FUNCTION_BLOCK FB_WinderSpeedControl
VAR_INPUT
    //==============================================================
    // ─────────────── MODE SELECTION / REFERENCES ───────────────
    //==============================================================
    groupSpeedAutoMan          : BOOL;  // TRUE = Auto, FALSE = Manual
    enableTorqueControl          : BOOL;  // TRUE = Auto, FALSE = Manual

    groupAutoSpeedMPM          : REAL;  // Auto speed reference [m/min]
    groupManualSpeedMPM        : REAL;  // Manual speed reference [m/min]
    groupRecoverSpeedCmd       : BOOL;  // Recover (temporary speed bump)
    groupRecoverIncrement      : REAL;  // Recover increment [m/min]

	
	torqueFeedback				: REAL;
    //==============================================================
    // ─────────────── DIAMETERS (mm) ───────────────
    //==============================================================
    diameter       : REAL;  // Diameter of group 1 master

    //==============================================================
    // ─────────────── CONFIGURATION / LIMITS ───────────────
    //==============================================================
    groupMasterMaxSpeedRPM     : REAL;  		// Max allowed master RPM
    rampUpRate					: REAL := 0.1;  // Ramp acceleration [RPM/s]
    rampDownRate				: REAL := 0.1;  // Ramp acceleration [RPM/s]
	
    state                      : INT;   // Machine state (5 = STOPPING)

    groupSpeedDifInc           : BOOL;  // Increment group speed offset
    groupSpeedDifDec           : BOOL;  // Decrement group speed offset
    groupSpeedDifLimLow        : REAL;  // Min offset [%]
    groupSpeedDifLimHigh       : REAL;  // Max offset [%]

    rampReset                  : BOOL;  // Reset ramp command
	
	
    torqueCtrlKp                   : REAL := 0.50;
    torqueCtrlTn                   : REAL := 5.0;
    torqueCtrlTv                   : REAL := 0.0;
	torqueDifLimitMin				: REAL := -3.0;
	torqueDifLimitMax				: REAL := 3.0;	
	
	
	
	
END_VAR


VAR_OUTPUT
    //==============================================================
    // ─────────────── FINAL DRIVE SPEEDS (RPM) ───────────────
    //==============================================================
    speedRefRPM    : REAL;


    //==============================================================
    // ─────────────── SURFACE SPEEDS (MPM) ───────────────
    //==============================================================
    group1MasterSpeedMPM       : REAL;


    //==============================================================
    // ─────────────── HANDOFF TO NEXT GROUP ───────────────
    //==============================================================
    nextGroupSpeedRefMPM       : REAL;
	speedDif					: REAL;
	
END_VAR


VAR
    //==============================================================
    // ─────────────── INTERNAL CALCULATION VARIABLES ───────────────
    //==============================================================
    masterMaxSpeedMPM          : REAL;
    baseCmdSpeedMPM            : REAL;
    cmdSpeedMPM                : REAL;
    targetRPM                  : REAL;
    rampTargetRPM              : REAL;
    baseMasterRefRPM           : REAL;
    groupSpeedOffset           : REAL;
    groupDeltaRatioAll         : REAL;
    upperLowerBiasRatio        : REAL;
    useRamp                    : BOOL;
    epsDiameter                : REAL := 0.001;

    // Gear ratios (set externally or calculated elsewhere)
    group1ToGroup1Slave1Ratio  : REAL := 1.0;
    group1ToGroup1Slave2Ratio  : REAL := 1.0;
    group1ToGroup2MasterRatio  : REAL := 1.0;
    group2ToGroup2Slave1Ratio  : REAL := 1.0;
    group2ToGroup2Slave2Ratio  : REAL := 1.0;

    // Function blocks
    instFB_Gen_SRamp           : FB_Gen_SRamp;
    speedOffsetPID   : REAL;  // Bias [%] between group1 and group2
 	instCTRL_PID_Group1TorqueTrim : CTRL_PID;
	rampActive: BOOL;
	enableTorqueControlOld: BOOL;
END_VAR

VAR_IN_OUT
	
	torqueSetpoint	: REAL;

END_VAR
VAR PERSISTENT
	
    instTUNE2_GroupSpeedDiff   : TUNE2;

END_VAR

//==============================================================
// IMPLEMENTATION
//==============================================================

//====================================================================
// ═══ CALL METHOD TO CALCULATE DIAMETER RATIOS ═════════════════════
//====================================================================
_CalculateGearRatios();

//--------------------------------------------------------------
// Calculate master max surface speed [m/min]
//--------------------------------------------------------------
masterMaxSpeedMPM := groupMasterMaxSpeedRPM * (PI * diameter) / 1000.0;


//--------------------------------------------------------------
// Determine base speed source (auto/manual) + Recover bump
//--------------------------------------------------------------
IF groupSpeedAutoMan THEN
    baseCmdSpeedMPM := groupAutoSpeedMPM;
ELSE
    baseCmdSpeedMPM := groupManualSpeedMPM;
END_IF;

IF groupRecoverSpeedCmd THEN
    cmdSpeedMPM := baseCmdSpeedMPM + groupRecoverIncrement;
ELSE
    cmdSpeedMPM := baseCmdSpeedMPM;
END_IF;


//--------------------------------------------------------------
// Convert MPM → target RPM for the master
//--------------------------------------------------------------
targetRPM := _Scale(
    X    := cmdSpeedMPM,
    I_LO := 0.0,
    I_HI := masterMaxSpeedMPM,
    O_LO := 0.0,
    O_HI := groupMasterMaxSpeedRPM);


//--------------------------------------------------------------
// Ramp handling
//--------------------------------------------------------------
IF state = 5 OR state = 0 THEN
    // STOPPING — force ramp down to zero speed
    rampTargetRPM := 0.0;

ELSIF state = 10 THEN
    // FAULT — clear ramp immediately to ensure no residual motion
    rampTargetRPM := 0.0;
//    rampReset     := TRUE;

ELSE
    // Normal operation — ramp follows target speed
    rampTargetRPM := targetRPM;
//    rampReset     := FALSE;
END_IF;

// Detect when a new target speed change requires ramping
IF NOT rampActive AND ABS(rampTargetRPM - baseMasterRefRPM) >= 1.0 THEN
   rampActive := TRUE; // Rising edge — ramp request detected
 
END_IF;

// Ramp function block execution
instFB_Gen_SRamp(
    X          := rampTargetRPM,
    A_UP       := MAX(0.0, rampUpRate),
    A_DN       := -MAX(0.0, rampDownRate),
    VU_MAX     := 1000.0,
    VD_MAX     := -1000.0,
    LIMIT_HIGH := groupMasterMaxSpeedRPM,
    RST        := rampReset);

// If ramping, update the baseMasterRefRPM from ramp output
IF rampActive THEN
    baseMasterRefRPM := instFB_Gen_SRamp.Y;

    // Automatically reset ramp flag when the ramp output reaches the target
    IF ABS(instFB_Gen_SRamp.Y - rampTargetRPM) <= 0.05 THEN
        rampActive := FALSE; // Ramp complete
    END_IF;

ELSE
    // No ramping required — direct assignment
    baseMasterRefRPM := rampTargetRPM;
END_IF;


(*
IF enableTorqueControl AND NOT enableTorqueControlOld THEN
	
	torqueSetpoint := torqueFeedback;
	
END_IF

enableTorqueControlOld := enableTorqueControl;
*)

IF NOT enableTorqueControl THEN
	
	instCTRL_PID_Group1TorqueTrim.LL := 0;
	instCTRL_PID_Group1TorqueTrim.LH := 0;
	
ELSE
	
	instCTRL_PID_Group1TorqueTrim.LL := torqueDifLimitMin;
	instCTRL_PID_Group1TorqueTrim.LH := torqueDifLimitMax;
	
END_IF



    instCTRL_PID_Group1TorqueTrim(
        ACT := torqueFeedback,
        SET := torqueSetpoint,
        MAN := FALSE,
        M_I := 0.0,
        RST := FALSE,
        KP  := torqueCtrlKp,
        TN  := torqueCtrlTn,
        TV  := torqueCtrlTv,
		SUP := 0.2,
        Y   => speedOffsetPID
    );

//--------------------------------------------------------------
// Operator offset (TUNE2 control)
//--------------------------------------------------------------
instTUNE2_GroupSpeedDiff(
    SET     := FALSE,
    SU      := groupSpeedDifInc,
    SD      := groupSpeedDifDec,
    RST     := FALSE,
    SS      := 0.01,
    FS      := 0.01,
    LIMIT_L := groupSpeedDifLimLow,
    LIMIT_H := groupSpeedDifLimHigh,
    Y       => groupSpeedOffset);

	
speedDif := groupSpeedOffset;
	
groupDeltaRatioAll  := 1.0 + ((speedOffsetPID + groupSpeedOffset) * 0.01);


//--------------------------------------------------------------
// Apply offsets + calculate all drive RPM references
//--------------------------------------------------------------
speedRefRPM := baseMasterRefRPM * groupDeltaRatioAll;


//--------------------------------------------------------------
// Convert RPM → MPM (surface speeds)
//--------------------------------------------------------------
group1MasterSpeedMPM := speedRefRPM * diameter * PI / 1000.0;


//--------------------------------------------------------------
// Suggest downstream handoff (group2 master surface speed)
//--------------------------------------------------------------
nextGroupSpeedRefMPM := group1MasterSpeedMPM;


//====================================================================
// ═══ PRIVATE METHOD — CALCULATE DIAMETER RATIOS ════════════════════
//====================================================================
METHOD PRIVATE _CalculateGearRatios
VAR_INPUT
END_VAR
;
END_METHOD

METHOD PRIVATE _Scale : REAL
VAR_INPUT
    X    : REAL;
    I_LO : REAL;
    I_HI : REAL;
    O_LO : REAL;
    O_HI : REAL;
END_VAR
IF I_LO = I_HI THEN
	_Scale := O_LO;
ELSE
	_Scale := (O_HI - O_LO) / (I_HI - I_LO) * (LIMIT(I_LO, X, I_HI) - I_LO) + O_LO;
END_IF;
END_METHOD

END_FUNCTION_BLOCK

(* stored: Version 1.1.0.1, ProductVersion 3.1.4024.15
   POU FB_WinderSpeedControl: Id {6103a0ee-9b7b-4a3e-900c-c4cdeacfa0ab}, SpecialFunc None
   Method _CalculateGearRatios: Id {e9f801e4-0b85-4ae6-beb8-eda86b67bfe2}
   Method _Scale: Id {198f4481-0ecf-47a0-8f4b-1cb851a6aa67} *)
